// TwinCAT 3 PLC project CodeAnalysis
// ProgramVersion: 3.1.4024.12
// project tree:
//   / POU.TcPOU
// I/O:
//   DEVICE Gerät 1 (EtherCAT), AmsNetId 10.0.2.15.2.1

// ---- POU.TcPOU
FUNCTION_BLOCK POU
VAR_INPUT
END_VAR
VAR_OUTPUT
END_VAR
VAR
	AddTwo: INT;
END_VAR

END_FUNCTION_BLOCK
